(* Logix 5000 project; controller START_STOP Emulate 5570 rev 30.12; software revision 30.00 *)

TASK MainTask (continuous, watchdog 500 ms) : MainProgram

MODULES
   Local : Emulate 5570 (ICP 2, rev 30.12)
      VIRTUAL_OUTPUTS : vendor 1 type 0 code 15 (ICP 4, rev 1.1, Output RPI 50 ms)
      VIRTUAL_INPUTS : vendor 1 type 0 code 15 (ICP 3, rev 1.1, Output RPI 50 ms)
END_MODULES

VAR_GLOBAL   (* controller tags *)
   CCR : BOOL;
   CE_DONE : BOOL;
   CM_DONE : BOOL;
   CT_RP_DN : BOOL;
   CVY_1 : ALIAS FOR Local:4:O.Data[0].7;
   CVY_12 : ALIAS FOR Local:4:O.Data[0].13;
   CVY_12_DN : BOOL;
   CVY_13 : ALIAS FOR Local:4:O.Data[0].14;
   CVY_13_DN : BOOL;
   CVY_1_2_DN : BOOL;
   CVY_2 : ALIAS FOR Local:4:O.Data[0].8;
   CVY_20 : ALIAS FOR Local:4:O.Data[0].4;
   CVY_21 : ALIAS FOR Local:4:O.Data[0].5;
   CVY_22 : ALIAS FOR Local:4:O.Data[0].6;
   CVY_22_DN : BOOL;
   CVY_3 : ALIAS FOR Local:4:O.Data[0].9;
   CVY_3_DN : BOOL;
   CVY_4 : ALIAS FOR Local:4:O.Data[0].10;
   CVY_4_DN : BOOL;
   CVY_5 : ALIAS FOR Local:4:O.Data[0].11;
   CVY_5_DN : BOOL;
   CVY_8 : ALIAS FOR Local:4:O.Data[0].3;
   CVY_8_DN : BOOL;
   DEL_1 : TIMER := (PRE := 1000);
   DEL_10 : TIMER := (PRE := 3000);
   DEL_11 : TIMER := (PRE := 1000);
   DEL_12 : TIMER := (PRE := 1000);
   DEL_15 : TIMER := (PRE := 1000);
   DEL_2 : TIMER := (PRE := 1000);
   DEL_3 : TIMER := (PRE := 1000);
   DEL_30 : TIMER := (PRE := 3000);
   DEL_4 : TIMER := (PRE := 1000);
   DEL_5 : TIMER := (PRE := 1000);
   DEL_7 : TIMER := (PRE := 1000);
   DEL_8 : TIMER := (PRE := 1000);
   DEL_9 : TIMER := (PRE := 1000);
   FIN_CE : BOOL;
   FIN_CM : BOOL;
   FIN_IR : BOOL;
   FIN_SP1 : BOOL;
   FIN_SP2 : BOOL;
   FIN_TL : BOOL;
   IR_DONE : BOOL;
   PB_CVY_1 : ALIAS FOR Local:3:I.Data[1].8;
   PB_CVY_12 : ALIAS FOR Local:3:I.Data[1].19;
   PB_CVY_13 : ALIAS FOR Local:3:I.Data[1].21;
   PB_CVY_2 : ALIAS FOR Local:3:I.Data[1].9;
   PB_CVY_22 : ALIAS FOR Local:3:I.Data[1].5;
   PB_CVY_3 : ALIAS FOR Local:3:I.Data[1].12;
   PB_CVY_4 : ALIAS FOR Local:3:I.Data[1].14;
   PB_CVY_5 : ALIAS FOR Local:3:I.Data[1].16;
   PB_CVY_8 : ALIAS FOR Local:3:I.Data[1].4;
   PRUEBA : BOOL;
   SNR_CVY_1 : ALIAS FOR Local:3:I.Data[1].10;
   SNR_CVY_12 : ALIAS FOR Local:3:I.Data[1].20;
   SNR_CVY_13 : ALIAS FOR Local:3:I.Data[1].22;
   SNR_CVY_2 : ALIAS FOR Local:3:I.Data[1].11;
   SNR_CVY_22 : ALIAS FOR Local:3:I.Data[1].7;
   SNR_CVY_3 : ALIAS FOR Local:3:I.Data[1].13;
   SNR_CVY_4 : ALIAS FOR Local:3:I.Data[1].15;
   SNR_CVY_5 : ALIAS FOR Local:3:I.Data[1].17;
   SNR_CVY_8 : ALIAS FOR Local:3:I.Data[1].6;
   SP1_DN : BOOL;
   SP2_DN : BOOL;
   SR1 : BOOL;
   SR13 : BOOL;
   SR18 : BOOL;
   SR19 : BOOL;
   SR2 : BOOL;
   SR27 : BOOL;
   SR28 : BOOL;
   SR3 : BOOL;
   SR33 : BOOL;
   SR34 : BOOL;
   SR35 : BOOL;
   SR4 : BOOL;
   SR5 : BOOL;
   SR6 : BOOL;
   SR7 : BOOL;
   SR8 : BOOL;
   SR9 : BOOL;
   Started : ALIAS FOR Local:4:O.Data[0].0;
   STP_g : ALIAS FOR Local:3:I.Data[1].1;
   STT_CE : ALIAS FOR Local:4:O.Data[0].16;
   STT_CM : ALIAS FOR Local:4:O.Data[0].15;
   STT_g : ALIAS FOR Local:3:I.Data[1].0;
   STT_IR : ALIAS FOR Local:4:O.Data[0].17;
   STT_SP1 : ALIAS FOR Local:4:O.Data[0].1;
   STT_SP2 : ALIAS FOR Local:4:O.Data[0].2;
   STT_TL : ALIAS FOR Local:4:O.Data[0].12;
   TF_1 : TIMER := (PRE := 2000);
   TF_10 : TIMER := (PRE := 2000);
   TF_2 : TIMER := (PRE := 2000);
   TF_3 : TIMER := (PRE := 2000);
   TF_4 : TIMER := (PRE := 2000);
   TF_5 : TIMER := (PRE := 2000);
   TF_6 : TIMER := (PRE := 2000);
   TF_7 : TIMER := (PRE := 2000);
   TF_8 : TIMER := (PRE := 2000);
   TF_9 : TIMER := (PRE := 2000);
   TL_DN : BOOL;
   TRN_10_DN : BOOL;
   TRN_11_DN : BOOL;
   TRN_29_DN : BOOL;
   TRN_33_DN : BOOL;
   TRN_34_DN : BOOL;
   TRN_35_DN : BOOL;
   TRN_3_DN : BOOL;
   TRN_4_DN : BOOL;
   TRN_8_DN : BOOL;
END_VAR

PROGRAM MainProgram   (* main routine MainRoutine *)

ROUTINE Encendido_CVY12   (* ladder *)
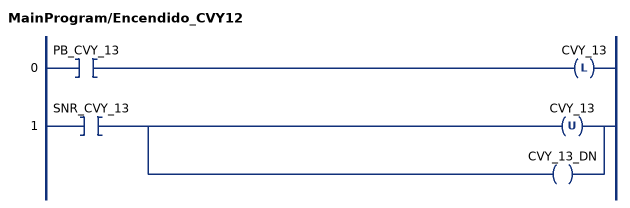
   0: XIC(PB_CVY_13)OTL(CVY_13);
   1: XIC(SNR_CVY_13)[OTU(CVY_13) ,OTE(CVY_13_DN) ];
END_ROUTINE

ROUTINE Encendido_CVY13   (* ladder *)
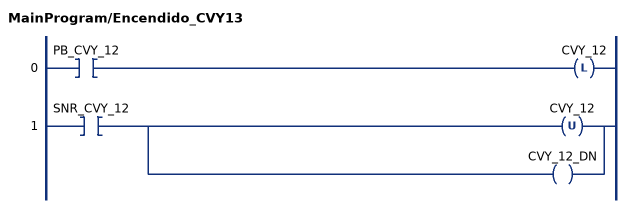
   0: XIC(PB_CVY_12)OTL(CVY_12);
   1: XIC(SNR_CVY_12)[OTU(CVY_12) ,OTE(CVY_12_DN) ];
END_ROUTINE

ROUTINE Encendido_CVY22   (* ladder *)
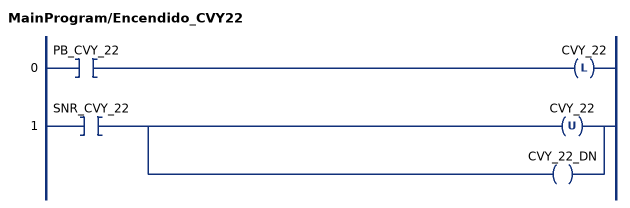
   0: XIC(PB_CVY_22)OTL(CVY_22);
   1: XIC(SNR_CVY_22)[OTU(CVY_22) ,OTE(CVY_22_DN) ];
END_ROUTINE

ROUTINE Encendido_CVY4   (* ladder *)
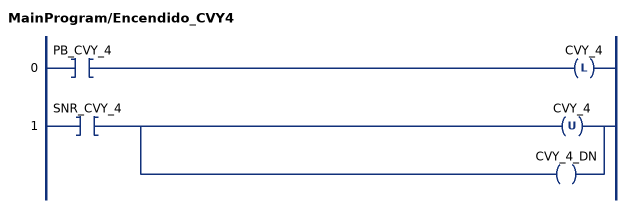
   0: XIC(PB_CVY_4)OTL(CVY_4);
   1: XIC(SNR_CVY_4)[OTU(CVY_4) ,OTE(CVY_4_DN) ];
END_ROUTINE

ROUTINE Encendido_CVY5   (* ladder *)
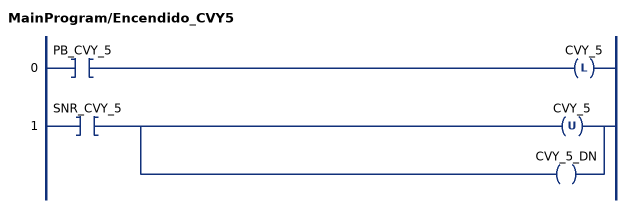
   0: XIC(PB_CVY_5)OTL(CVY_5);
   1: XIC(SNR_CVY_5)[OTU(CVY_5) ,OTE(CVY_5_DN) ];
END_ROUTINE

ROUTINE Encendido_CVY8   (* ladder *)
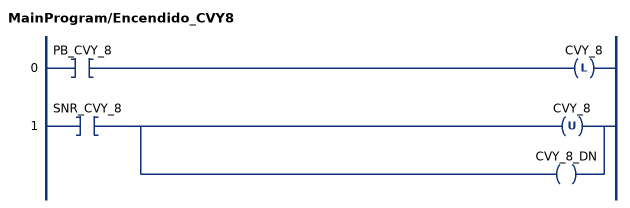
   0: XIC(PB_CVY_8)OTL(CVY_8);
   1: XIC(SNR_CVY_8)[OTU(CVY_8) ,OTE(CVY_8_DN) ];
END_ROUTINE

ROUTINE Inicio_Corte_reposabrazos   (* ladder *)
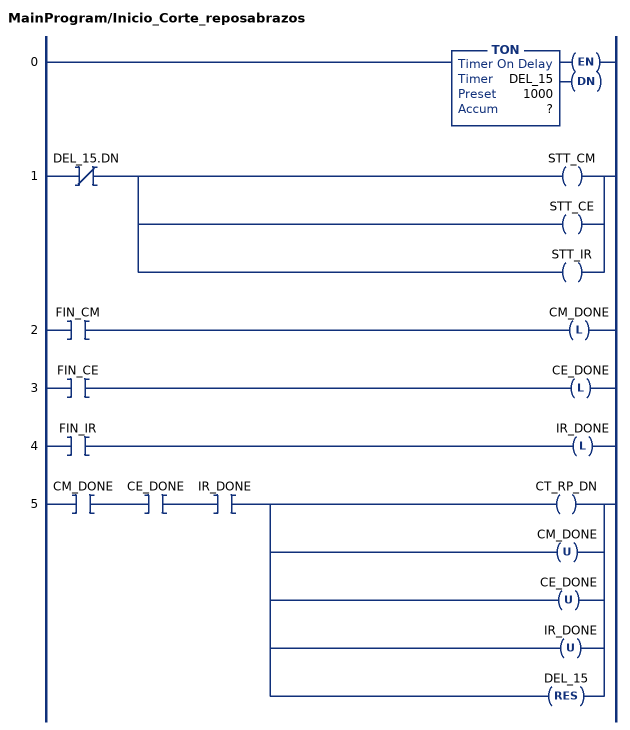
   0: TON(DEL_15,?,?);
   1: XIO(DEL_15.DN)[OTE(STT_CM) ,OTE(STT_CE) ,OTE(STT_IR) ];
   2: XIC(FIN_CM)OTL(CM_DONE);
   3: XIC(FIN_CE)OTL(CE_DONE);
   4: XIC(FIN_IR)OTL(IR_DONE);
   5: XIC(CM_DONE)XIC(CE_DONE)XIC(IR_DONE)[OTE(CT_RP_DN) ,OTU(CM_DONE) ,OTU(CE_DONE) ,OTU(IR_DONE) ,RES(DEL_15) ];
END_ROUTINE

ROUTINE Inicio_Soplado   (* ladder *)
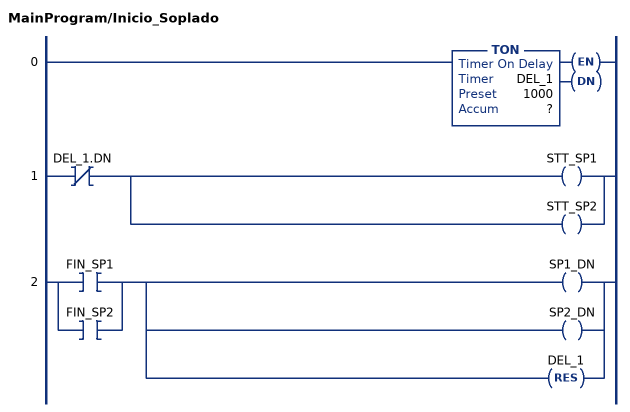
   0: TON(DEL_1,?,?);
   1: XIO(DEL_1.DN)[OTE(STT_SP1) ,OTE(STT_SP2) ];
   2: [XIC(FIN_SP1) ,XIC(FIN_SP2) ][OTE(SP1_DN) ,OTE(SP2_DN) ,RES(DEL_1) ];
END_ROUTINE

ROUTINE Inicio_Taladrado   (* ladder *)
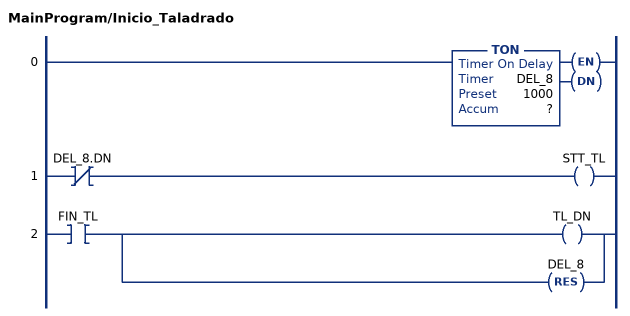
   0: TON(DEL_8,?,?);
   1: XIO(DEL_8.DN)OTE(STT_TL);
   2: XIC(FIN_TL)[OTE(TL_DN) ,RES(DEL_8) ];
END_ROUTINE

ROUTINE MainRoutine   (* ladder *)
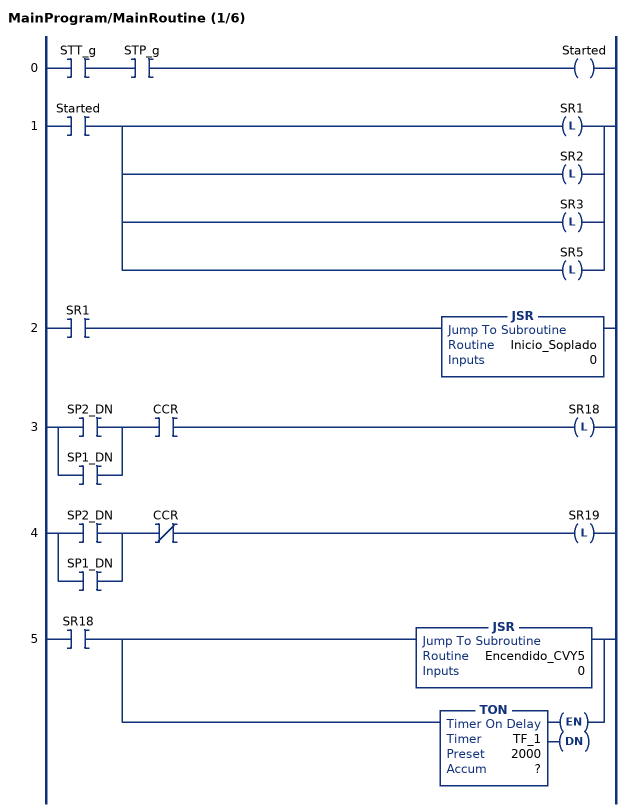
   0: XIC(STT_g)XIC(STP_g)OTE(Started);
   1: XIC(Started)[OTL(SR1) ,OTL(SR2) ,OTL(SR3) ,OTL(SR5) ];
   2: XIC(SR1)JSR(Inicio_Soplado,0);
   3: [XIC(SP2_DN) ,XIC(SP1_DN) ]XIC(CCR)OTL(SR18);
   4: [XIC(SP2_DN) ,XIC(SP1_DN) ]XIO(CCR)OTL(SR19);
   5: XIC(SR18)[JSR(Encendido_CVY5,0) ,TON(TF_1,?,?) ];
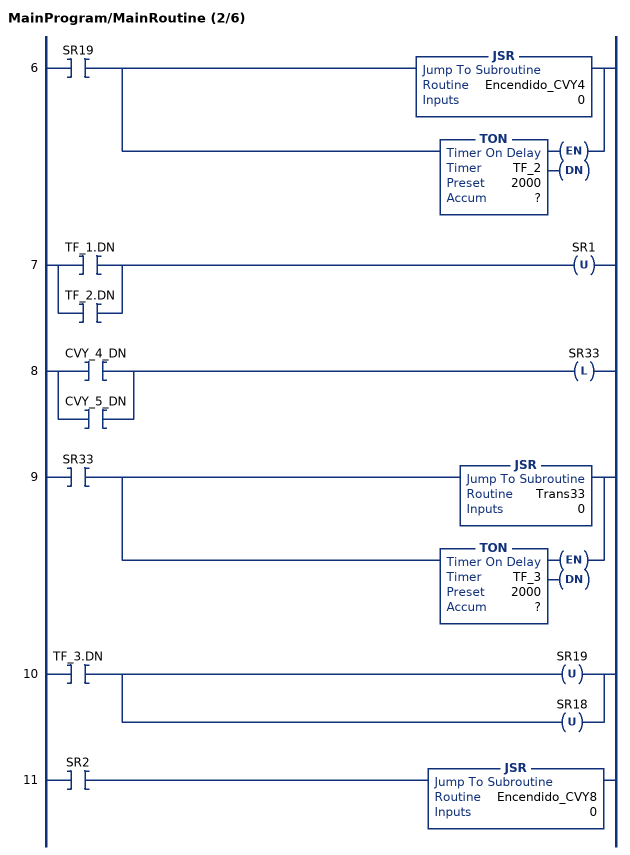
   6: XIC(SR19)[JSR(Encendido_CVY4,0) ,TON(TF_2,?,?) ];
   7: [XIC(TF_1.DN) ,XIC(TF_2.DN) ]OTU(SR1);
   8: [XIC(CVY_4_DN) ,XIC(CVY_5_DN) ]OTL(SR33);
   9: XIC(SR33)[JSR(Trans33,0) ,TON(TF_3,?,?) ];
   10: XIC(TF_3.DN)[OTU(SR19) ,OTU(SR18) ];
   11: XIC(SR2)JSR(Encendido_CVY8,0);
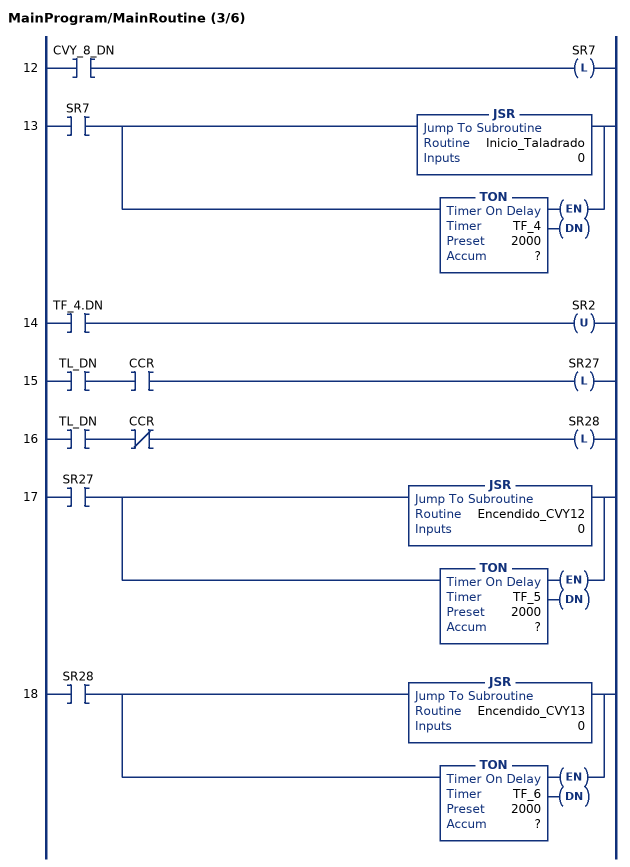
   12: XIC(CVY_8_DN)OTL(SR7);
   13: XIC(SR7)[JSR(Inicio_Taladrado,0) ,TON(TF_4,?,?) ];
   14: XIC(TF_4.DN)OTU(SR2);
   15: XIC(TL_DN)XIC(CCR)OTL(SR27);
   16: XIC(TL_DN)XIO(CCR)OTL(SR28);
   17: XIC(SR27)[JSR(Encendido_CVY12,0) ,TON(TF_5,?,?) ];
   18: XIC(SR28)[JSR(Encendido_CVY13,0) ,TON(TF_6,?,?) ];
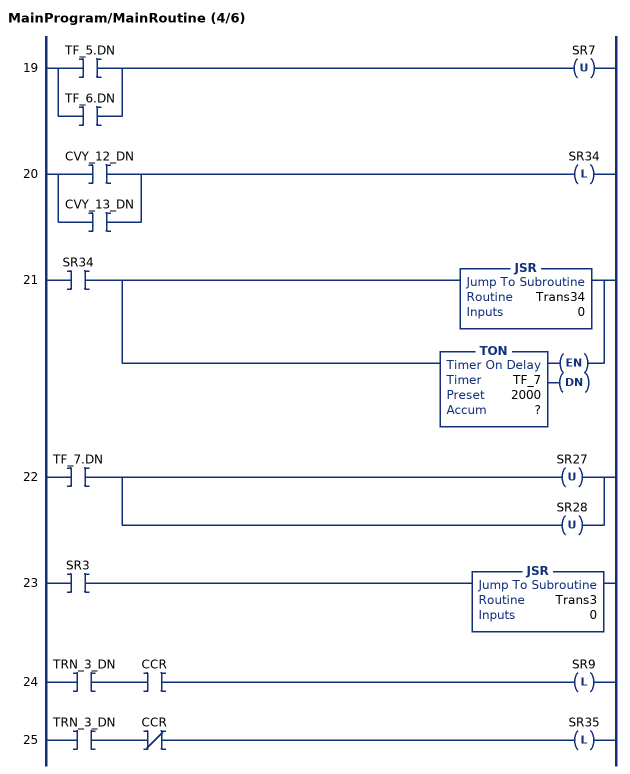
   19: [XIC(TF_5.DN) ,XIC(TF_6.DN) ]OTU(SR7);
   20: [XIC(CVY_12_DN) ,XIC(CVY_13_DN) ]OTL(SR34);
   21: XIC(SR34)[JSR(Trans34,0) ,TON(TF_7,?,?) ];
   22: XIC(TF_7.DN)[OTU(SR27) ,OTU(SR28) ];
   23: XIC(SR3)JSR(Trans3,0);
   24: XIC(TRN_3_DN)XIC(CCR)OTL(SR9);
   25: XIC(TRN_3_DN)XIO(CCR)OTL(SR35);
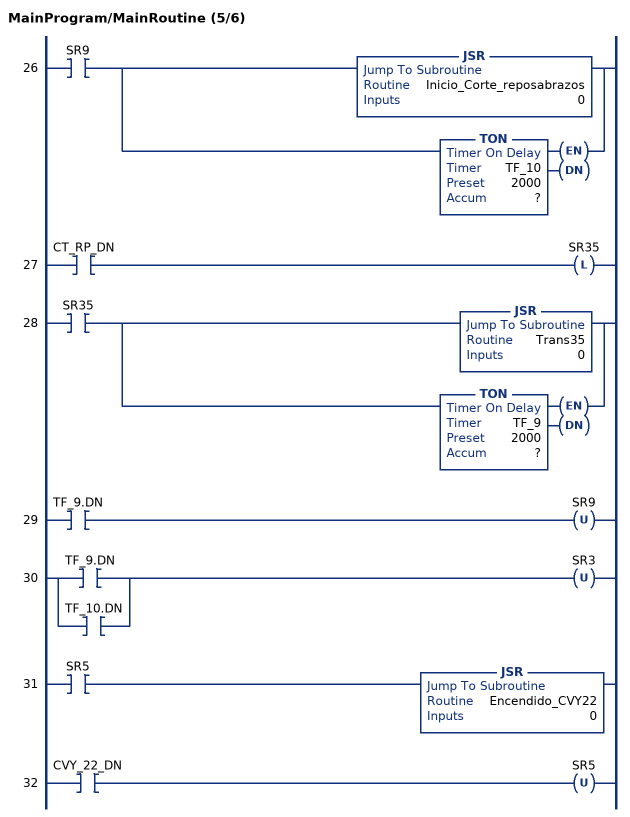
   26: XIC(SR9)[JSR(Inicio_Corte_reposabrazos,0) ,TON(TF_10,?,?) ];
   27: XIC(CT_RP_DN)OTL(SR35);
   28: XIC(SR35)[JSR(Trans35,0) ,TON(TF_9,?,?) ];
   29: XIC(TF_9.DN)OTU(SR9);
   30: [XIC(TF_9.DN) ,XIC(TF_10.DN) ]OTU(SR3);
   31: XIC(SR5)JSR(Encendido_CVY22,0);
   32: XIC(CVY_22_DN)OTU(SR5);
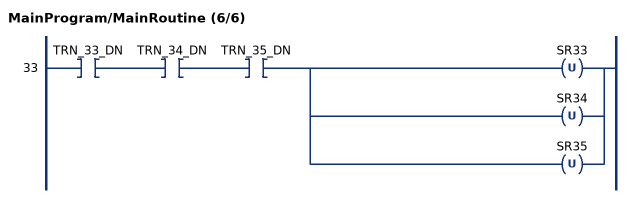
   33: XIC(TRN_33_DN)XIC(TRN_34_DN)XIC(TRN_35_DN)[OTU(SR33) ,OTU(SR34) ,OTU(SR35) ];
END_ROUTINE

ROUTINE Trans3   (* ladder *)
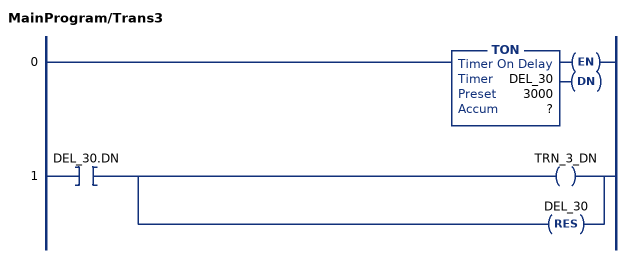
   0: TON(DEL_30,?,?);
   1: XIC(DEL_30.DN)[OTE(TRN_3_DN) ,RES(DEL_30) ];
END_ROUTINE

ROUTINE Trans33   (* ladder *)
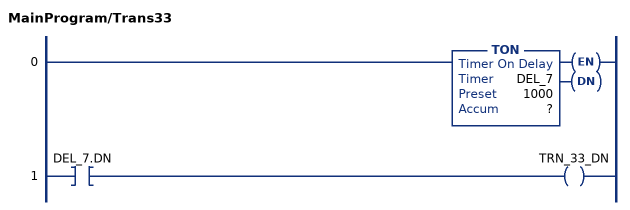
   0: TON(DEL_7,?,?);
   1: XIC(DEL_7.DN)OTE(TRN_33_DN);
END_ROUTINE

ROUTINE Trans34   (* ladder *)
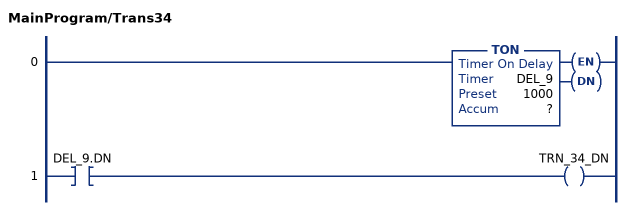
   0: TON(DEL_9,?,?);
   1: XIC(DEL_9.DN)OTE(TRN_34_DN);
END_ROUTINE

ROUTINE Trans35   (* ladder *)
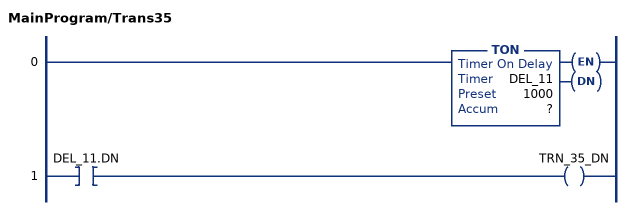
   0: TON(DEL_11,?,?);
   1: XIC(DEL_11.DN)OTE(TRN_35_DN);
END_ROUTINE
END_PROGRAM
